// Automatisch erzeugter Code: NICHT EDITIEREN
FUNCTION CheckBounds : DINT
VAR_INPUT
	index, lower, upper: DINT;
END_VAR

// Automatisch erzeugter Code: Es handelt sich hierbei um einen Implementierungsvorschlag.
{noflow}
IF  index < lower THEN
	CheckBounds := lower;
ELSIF  index > upper THEN
	CheckBounds := upper;
ELSE  
	CheckBounds := index;
END_IF
{flow}

END_FUNCTION

(* stored: Version 1.1.0.1, ProductVersion 3.1.4024.10
   POU CheckBounds: Id {110b8f3c-03aa-45d3-b75f-1e66b870a459}, SpecialFunc CheckBounds *)
